FUNCTION Convert_ULINT_TO_LWORD : Hresult
VAR_INPUT
	in : ULINT;
	out : REFERENCE TO LWORD;
END_VAR
VAR
	converted : LWORD;
END_VAR

converted := ULINT_TO_LWORD(in);

IF (LWORD_TO_ULINT(converted) <> in) THEN
	Convert_ULINT_TO_LWORD := INCOMPATIBLE;
	RETURN;
END_IF

out := converted;

END_FUNCTION

(* stored: Version 1.1.0.1, ProductVersion 3.1.4024.12
   POU Convert_ULINT_TO_LWORD: Id {620479a9-b7a3-4166-8700-054cdc476a82}, SpecialFunc None *)
